{attribute 'linkalways'} 
{attribute 'no_explicit_call' := 'This FB is a CLASS and must be accessed using methods or properties'}
{attribute 'enable_dynamic_creation'}
FUNCTION_BLOCK FINAL NOT_DINT EXTENDS Node
VAR
	in : _DINT(0);
	out : _DINT(0);
END_VAR

METHOD PUBLIC Clone : I_Node
VAR
	pNode : POINTER TO NOT_DINT;
END_VAR
pNode := __NEW(NOT_DINT);
Clone := pNode^;
END_METHOD

METHOD FB_init : BOOL
VAR_INPUT
	bInitRetains : BOOL; // if TRUE, the retain variables are initialized (warm start / cold start)
	bInCopyCode : BOOL;  // if TRUE, the instance afterwards gets moved into the copy code (online change)
END_VAR
AddInput('in',THIS^.in);
AddOutput('out', THIS^.out);
END_METHOD

METHOD PROTECTED OnExecute
VAR
END_VAR
out.Value := NOT in.Value;
END_METHOD

END_FUNCTION_BLOCK

(* stored: Version 1.1.0.1, ProductVersion 3.1.4024.15
   POU NOT_DINT: Id {72d289ca-c6c7-4a58-a4f2-eabea8090f87}, SpecialFunc None
   Folder Constructor: Id {bcd6c11b-e0b6-4ca9-8c12-75400981cf90}
   Method Clone: Id {f5b0b6bc-3d1c-4fa9-9d42-9c74d4bfdd2d}
   Method FB_init: Id {024d3402-9415-4fe9-85a1-6cf76edbba5f}
   Method OnExecute: Id {0eef9107-273f-45b8-b726-b36c44877adc} *)
